{attribute 'qualified_only'}
VAR_GLOBAL
	DI_BtnYellow    AT %I* : BOOL;
    DI_BtnBlue      AT %I* : BOOL;
	DI_BtnGreen     AT %I* : BOOL;
    
    DO_LampRed      AT %Q* : BOOL;
    DO_LampGreen    AT %Q* : BOOL;
	DO_LampOrange   AT %Q* : BOOL;
END_VAR

(* stored: Version 1.1.0.1, ProductVersion 3.1.4024.9
   GVL GVL_IO: Id {ec9c2cea-2085-4faa-836d-81012fcaa7fd} *)
